PROGRAM MAIN
VAR
END_VAR

END_PROGRAM

(* stored: Version 1.1.0.1
   POU MAIN: Id {a5319346-ab93-4f3a-a621-85d2937c3e0a} *)
